(* PLC project Unnamed, Unknown Unnamed 1 *)
(* stored: creationDateTime 2022-02-24T14:40:38, modificationDateTime 2022-08-17T12:03:17 *)

PROGRAM Arduino_Cloud
  VAR
    TON0 : TON;
    TOF0 : TOF;
    oscillator_pulse : BOOL;
    CTU0 : CTU;
    CTU_reset : BOOL;
  END_VAR
  VAR
    minute_count AT %QW0 : INT;
  END_VAR
  VAR
    CLOUD_BEGIN0 : CLOUD_BEGIN;
    CLOUD_ADD_DINT0 : CLOUD_ADD_DINT;
    CLOUD_ADD_BOOL0 : CLOUD_ADD_BOOL;
    TON1 : TON;
    time_lapsed : REAL;
    time_lapsed_reset : BOOL;
    CLOUD_ADD_REAL0 : CLOUD_ADD_REAL;
  END_VAR
  VAR  (* added by the conversion: wires and edge detectors of the diagram *)
    R_TRIG1 : R_TRIG;
  END_VAR

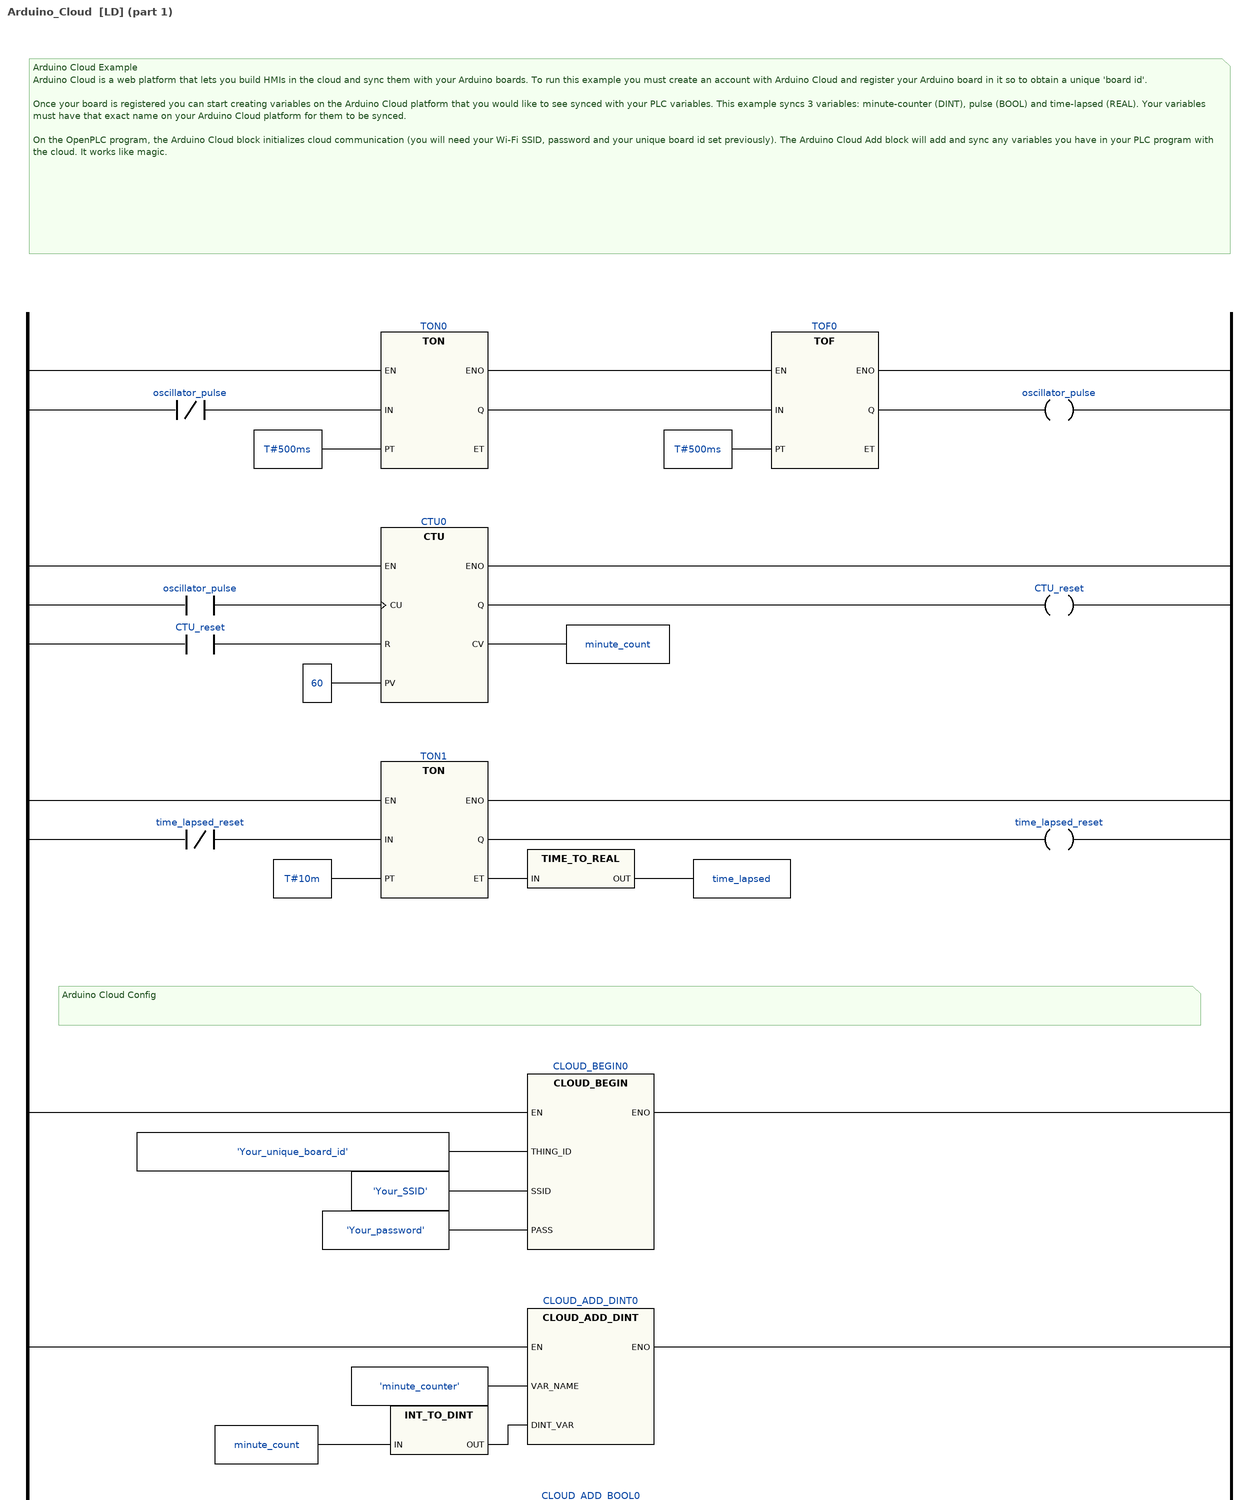
(* LD diagram, written out as Structured Text *)
(* Arduino Cloud Example
Arduino Cloud is a web platform that lets you build HMIs in the cloud and sync them with your Arduino boards. To run this example you must create an account with Arduino Cloud and register your Arduino board in it so to obtain a unique 'board id'.

Once your board is registered you can start creating variables on the Arduino Cloud platform that you would like to see synced with your PLC variables. This example syncs 3 variables: minute-counter (DINT), pulse (BOOL) and time-lapsed (REAL). Your variables must have that exact name on your Arduino Cloud platform for them to be synced.

On the OpenPLC program, the Arduino Cloud block initializes cloud communication (you will need your Wi-Fi SSID, password and your unique board id set previously). The Arduino Cloud Add block will add and sync any variables you have in your PLC program with the cloud. It works like magic. *)
TON0(IN := NOT oscillator_pulse, PT := T#500ms);
TOF0(EN := TON0.ENO, IN := TON0.Q, PT := T#500ms);
oscillator_pulse := TOF0.Q;
R_TRIG1(CLK := oscillator_pulse);
CTU0(CU := R_TRIG1.Q, R := CTU_reset, PV := 60);
CTU_reset := CTU0.Q;
minute_count := CTU0.CV;
TON1(IN := NOT time_lapsed_reset, PT := T#10m);
time_lapsed_reset := TON1.Q;
time_lapsed := TIME_TO_REAL(TON1.ET);
(* Arduino Cloud Config *)
CLOUD_BEGIN0(THING_ID := 'Your_unique_board_id', SSID := 'Your_SSID', PASS := 'Your_password');
CLOUD_ADD_DINT0(VAR_NAME := 'minute_counter', DINT_VAR := INT_TO_DINT(minute_count));
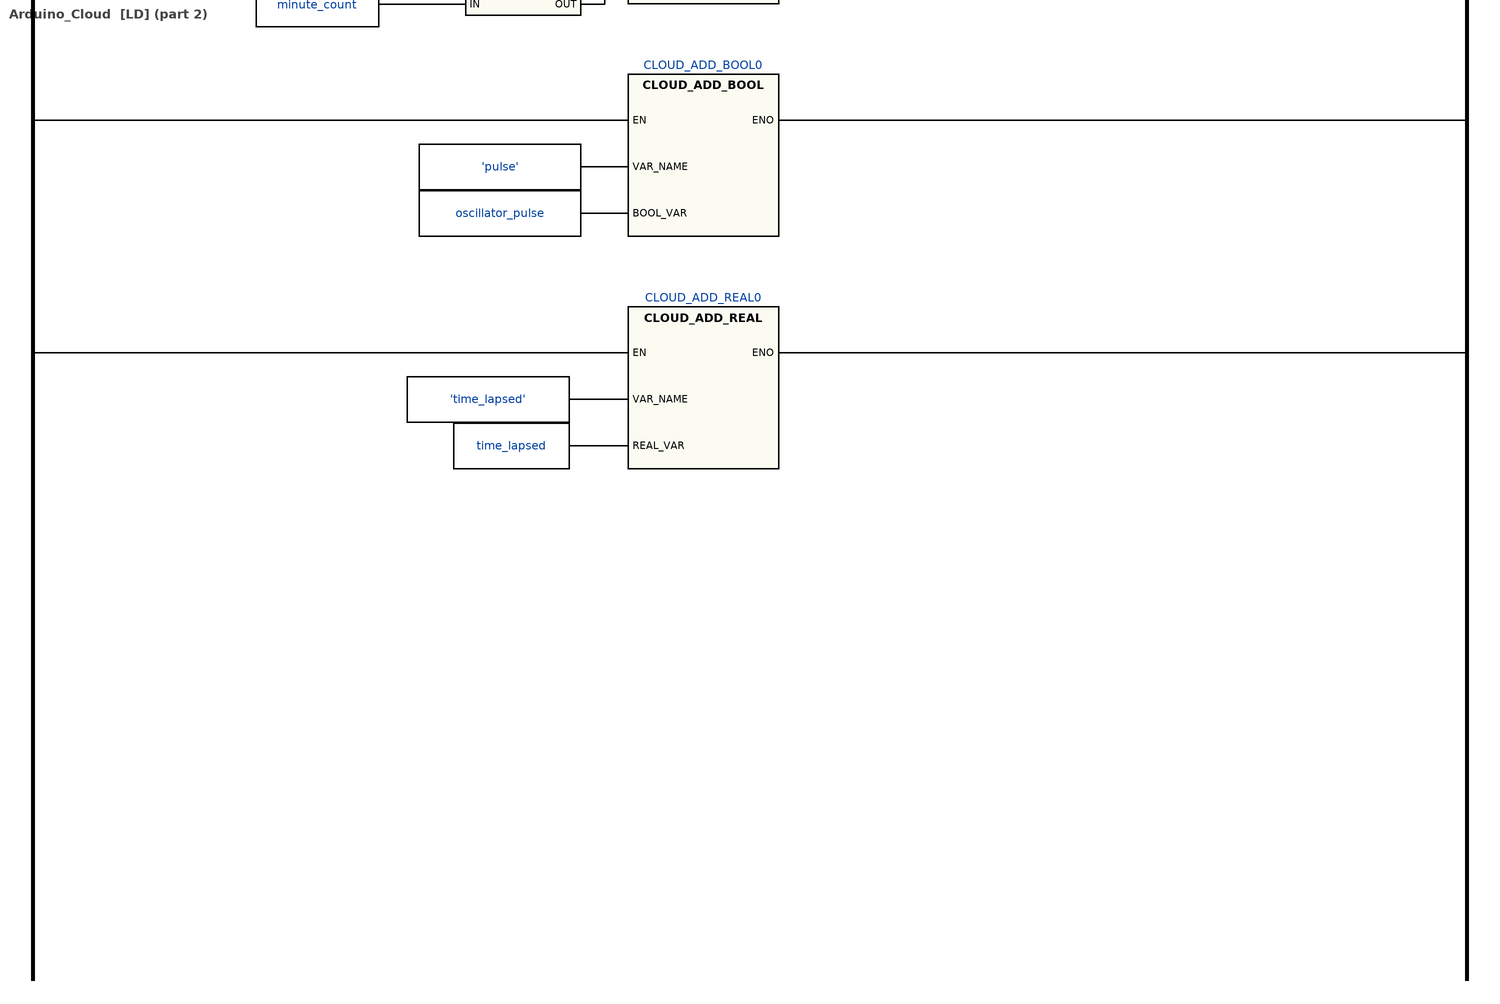
CLOUD_ADD_BOOL0(VAR_NAME := 'pulse', BOOL_VAR := oscillator_pulse);
CLOUD_ADD_REAL0(VAR_NAME := 'time_lapsed', REAL_VAR := time_lapsed);
END_PROGRAM

CONFIGURATION Config0
  RESOURCE Res0 ON PLC
    TASK task0(INTERVAL := T#20ms, PRIORITY := 0);
    PROGRAM instance0 WITH task0 : Arduino_Cloud;
  END_RESOURCE
END_CONFIGURATION
